// TIA Portal V18 export
ORGANIZATION_BLOCK "15-Slope"   // OB128, LAD, ProgramCycle
TITLE = "Main Program Sweep (Cycle)"
{ S7_Optimized_Access := 'TRUE' }
VERSION : 0.1
// stored: AutoNumber true, IsIECCheckEnabled false, SetENOAutomatically false
   VAR_INPUT
      Initial_Call : Bool;   // Initial call of this OB
      Remanence : Bool;   // =True, if remanent data are available
   END_VAR
   VAR_TEMP
      "Temp_1 (NormScale) Wire" : Real;
      "Temp_2 (NormScale) Inclanation" : Real;
      Temp_3 : Real;
      "Temp_4 (Radyan)" : Real;
      Temp_5 : Real;
      "Temp-6 AnimasyonNorm" : Real;
   END_VAR
BEGIN

REGION Network 1: Slope Angle
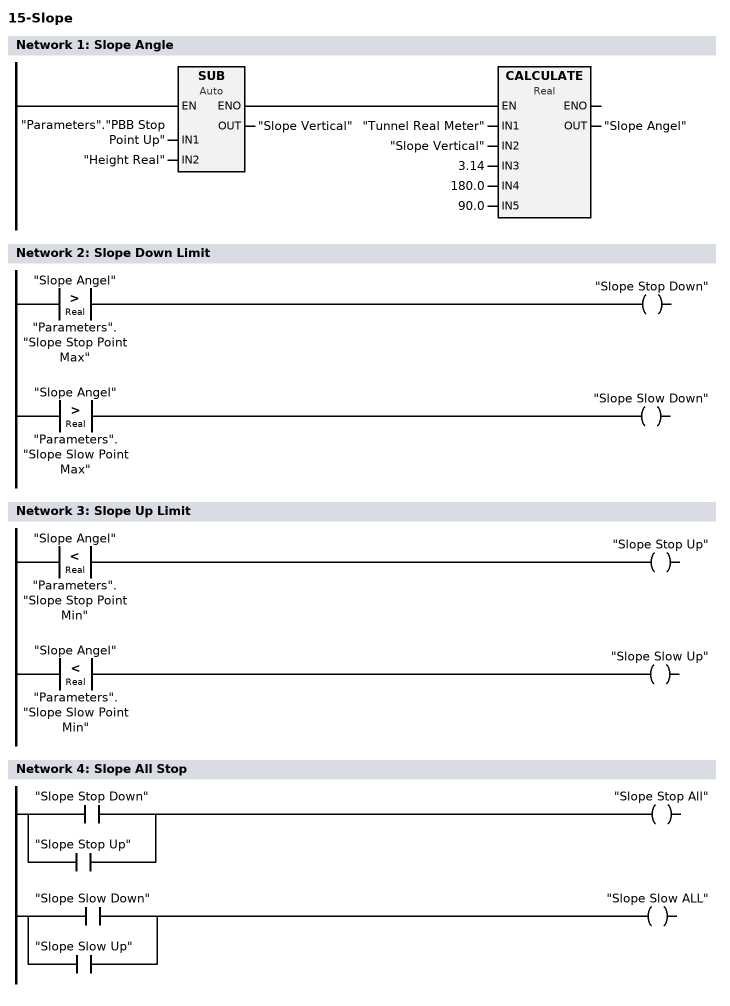
   RUNG wire#powerrail
      Sub(in1 := "Parameters"."PBB Stop Point Up", in2 := "Height Real", out => "Slope Vertical")
      { S7_Templates := "SrcType := Real"; S7_Expression := "IN5 -((ACOS(IN2 / IN1) *IN4) / IN3)" } Calculate(in1 := "Tunnel Real Meter", in2 := "Slope Vertical", in3 := 3.14, in4 := 180.0, in5 := 90.0, out => "Slope Angel")
   END_RUNG
   // the same network as SCL:
   "Slope Vertical" := "Parameters"."PBB Stop Point Up" - "Height Real";
   "Slope Angel" := 90.0 -((ACOS("Slope Vertical" / "Tunnel Real Meter") *180.0) / 3.14);
END_REGION

REGION Network 2: Slope Down Limit
   RUNG wire#powerrail
      { S7_Templates := "SrcType := Real" } GT_Contact(in1 := "Slope Angel", in2 := "Parameters"."Slope Stop Point Max")
      Coil( "Slope Stop Down" )
   END_RUNG
   RUNG wire#powerrail
      { S7_Templates := "SrcType := Real" } GT_Contact(in1 := "Slope Angel", in2 := "Parameters"."Slope Slow Point Max")
      Coil( "Slope Slow Down" )
   END_RUNG
   // the same network as SCL:
   "Slope Stop Down" := "Slope Angel" > "Parameters"."Slope Stop Point Max";
   "Slope Slow Down" := "Slope Angel" > "Parameters"."Slope Slow Point Max";
END_REGION

REGION Network 3: Slope Up Limit
   RUNG wire#powerrail
      { S7_Templates := "SrcType := Real" } LT_Contact(in1 := "Slope Angel", in2 := "Parameters"."Slope Stop Point Min")
      Coil( "Slope Stop Up" )
   END_RUNG
   RUNG wire#powerrail
      { S7_Templates := "SrcType := Real" } LT_Contact(in1 := "Slope Angel", in2 := "Parameters"."Slope Slow Point Min")
      Coil( "Slope Slow Up" )
   END_RUNG
   // the same network as SCL:
   "Slope Stop Up" := "Slope Angel" < "Parameters"."Slope Stop Point Min";
   "Slope Slow Up" := "Slope Angel" < "Parameters"."Slope Slow Point Min";
END_REGION

REGION Network 4: Slope All Stop
   RUNG wire#powerrail
      Contact( "Slope Stop Down" )
      wire#w1
      Coil( "Slope Stop All" )
   END_RUNG
   RUNG wire#powerrail
      Contact( "Slope Stop Up" )
   END_RUNG wire#w1
   RUNG wire#powerrail
      Contact( "Slope Slow Down" )
      wire#w2
      Coil( "Slope Slow ALL" )
   END_RUNG
   RUNG wire#powerrail
      Contact( "Slope Slow Up" )
   END_RUNG wire#w2
   // the same network as SCL:
   "Slope Stop All" := "Slope Stop Down" OR "Slope Stop Up";
   "Slope Slow ALL" := "Slope Slow Down" OR "Slope Slow Up";
END_REGION
END_ORGANIZATION_BLOCK
